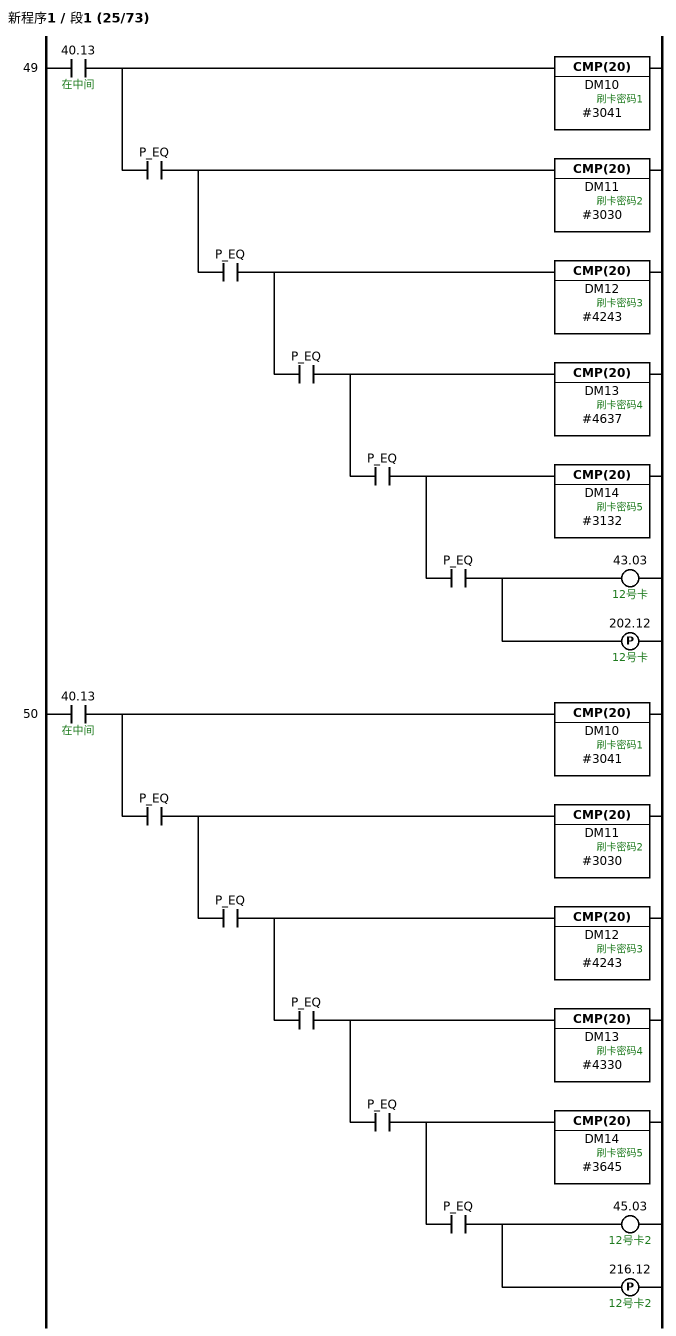
; [picture p24: 新程序1 / 段1, rungs 49-50]
; rung 49
LD 40.13  ; 在中间
CMP(20) DM10 #3041  ; 刷卡密码1
AND P_EQ
CMP(20) DM11 #3030  ; 刷卡密码2
AND P_EQ
CMP(20) DM12 #4243  ; 刷卡密码3
AND P_EQ
CMP(20) DM13 #4637  ; 刷卡密码4
AND P_EQ
CMP(20) DM14 #3132  ; 刷卡密码5
AND P_EQ
OUT 43.03  ; 12号卡
DIFU(13) 202.12  ; 12号卡
; rung 50
LD 40.13  ; 在中间
CMP(20) DM10 #3041  ; 刷卡密码1
AND P_EQ
CMP(20) DM11 #3030  ; 刷卡密码2
AND P_EQ
CMP(20) DM12 #4243  ; 刷卡密码3
AND P_EQ
CMP(20) DM13 #4330  ; 刷卡密码4
AND P_EQ
CMP(20) DM14 #3645  ; 刷卡密码5
AND P_EQ
OUT 45.03  ; 12号卡2
DIFU(13) 216.12  ; 12号卡2

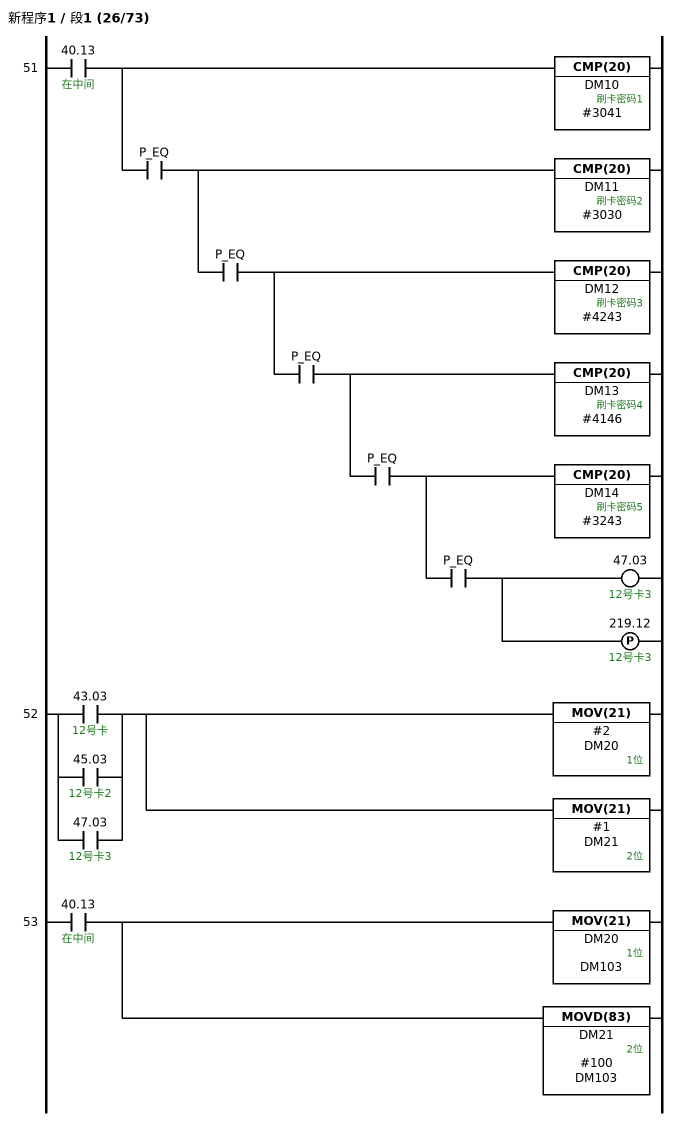
; rung 51
LD 40.13  ; 在中间
CMP(20) DM10 #3041  ; 刷卡密码1
AND P_EQ
CMP(20) DM11 #3030  ; 刷卡密码2
AND P_EQ
CMP(20) DM12 #4243  ; 刷卡密码3
AND P_EQ
CMP(20) DM13 #4146  ; 刷卡密码4
AND P_EQ
CMP(20) DM14 #3243  ; 刷卡密码5
AND P_EQ
OUT 47.03  ; 12号卡3
DIFU(13) 219.12  ; 12号卡3
; rung 52
LD 43.03  ; 12号卡
OR 45.03  ; 12号卡2
OR 47.03  ; 12号卡3
MOV(21) #2 DM20  ; 1位
MOV(21) #1 DM21  ; 2位
; rung 53
LD 40.13  ; 在中间
MOV(21) DM20 DM103  ; 1位
MOVD(83) DM21 #100 DM103  ; 2位

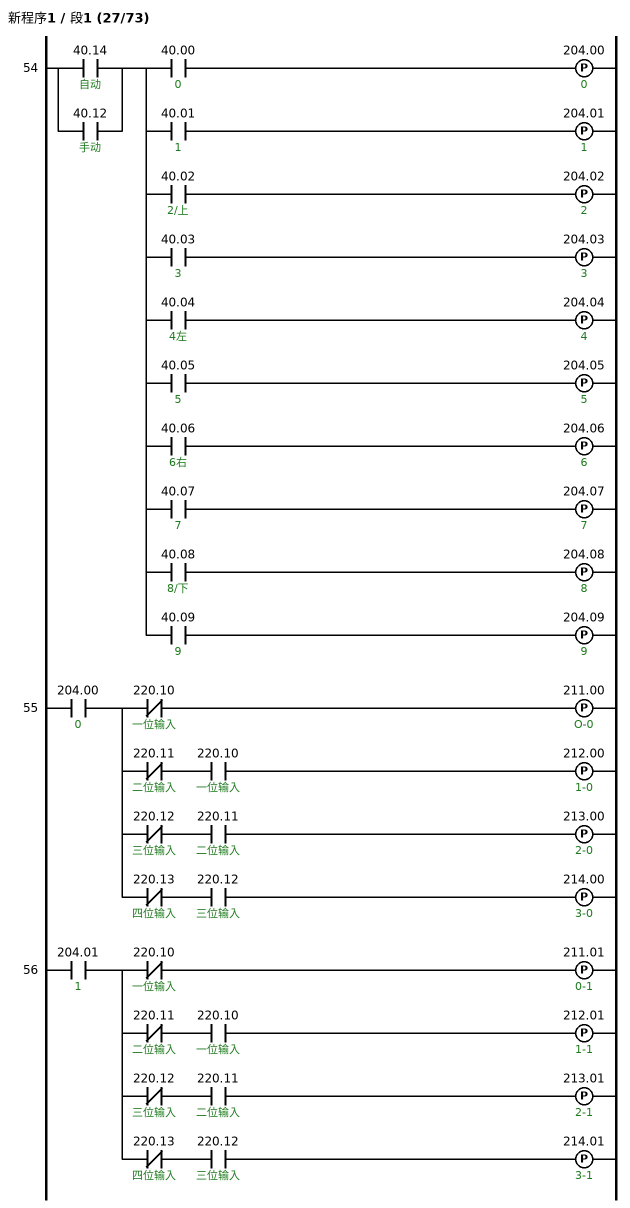
; rung 54
LD 40.14  ; 自动
OR 40.12  ; 手动
OUT TR0
AND 40.00  ; 0
DIFU(13) 204.00  ; 0
LD TR0
AND 40.01  ; 1
DIFU(13) 204.01  ; 1
LD TR0
AND 40.02  ; 2/上
DIFU(13) 204.02  ; 2
LD TR0
AND 40.03  ; 3
DIFU(13) 204.03  ; 3
LD TR0
AND 40.04  ; 4左
DIFU(13) 204.04  ; 4
LD TR0
AND 40.05  ; 5
DIFU(13) 204.05  ; 5
LD TR0
AND 40.06  ; 6右
DIFU(13) 204.06  ; 6
LD TR0
AND 40.07  ; 7
DIFU(13) 204.07  ; 7
LD TR0
AND 40.08  ; 8/下
DIFU(13) 204.08  ; 8
LD TR0
AND 40.09  ; 9
DIFU(13) 204.09  ; 9
; rung 55
LD 204.00  ; 0
OUT TR0
ANDNOT 220.10  ; 一位输入
DIFU(13) 211.00  ; O-0
LD TR0
ANDNOT 220.11  ; 二位输入
AND 220.10  ; 一位输入
DIFU(13) 212.00  ; 1-0
LD TR0
ANDNOT 220.12  ; 三位输入
AND 220.11  ; 二位输入
DIFU(13) 213.00  ; 2-0
LD TR0
ANDNOT 220.13  ; 四位输入
AND 220.12  ; 三位输入
DIFU(13) 214.00  ; 3-0
; rung 56
LD 204.01  ; 1
OUT TR0
ANDNOT 220.10  ; 一位输入
DIFU(13) 211.01  ; 0-1
LD TR0
ANDNOT 220.11  ; 二位输入
AND 220.10  ; 一位输入
DIFU(13) 212.01  ; 1-1
LD TR0
ANDNOT 220.12  ; 三位输入
AND 220.11  ; 二位输入
DIFU(13) 213.01  ; 2-1
LD TR0
ANDNOT 220.13  ; 四位输入
AND 220.12  ; 三位输入
DIFU(13) 214.01  ; 3-1

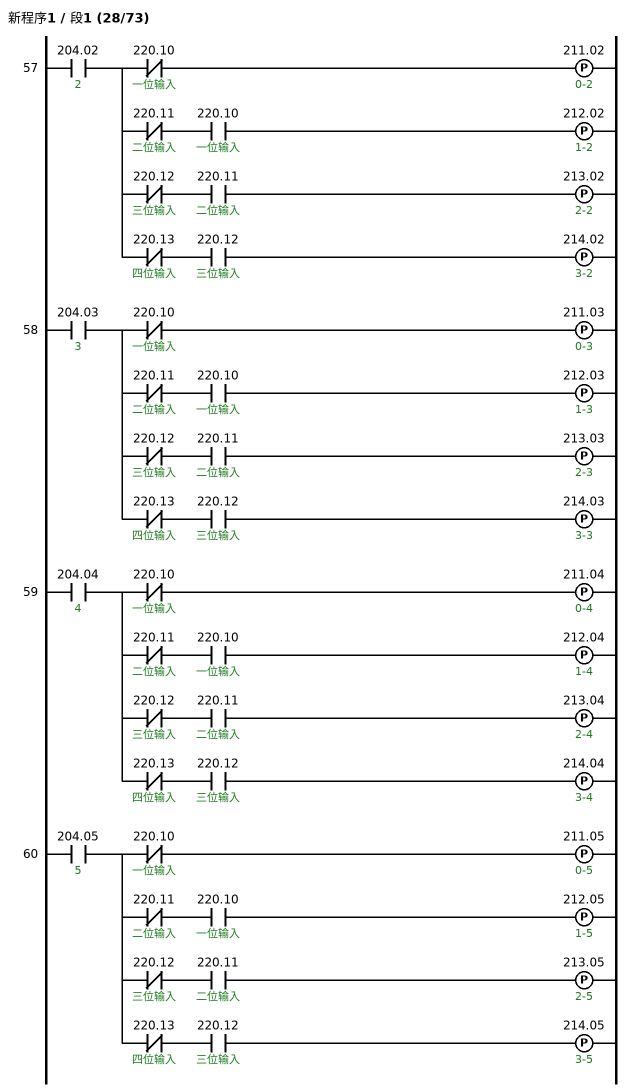
; rung 57
LD 204.02  ; 2
OUT TR0
ANDNOT 220.10  ; 一位输入
DIFU(13) 211.02  ; 0-2
LD TR0
ANDNOT 220.11  ; 二位输入
AND 220.10  ; 一位输入
DIFU(13) 212.02  ; 1-2
LD TR0
ANDNOT 220.12  ; 三位输入
AND 220.11  ; 二位输入
DIFU(13) 213.02  ; 2-2
LD TR0
ANDNOT 220.13  ; 四位输入
AND 220.12  ; 三位输入
DIFU(13) 214.02  ; 3-2
; rung 58
LD 204.03  ; 3
OUT TR0
ANDNOT 220.10  ; 一位输入
DIFU(13) 211.03  ; 0-3
LD TR0
ANDNOT 220.11  ; 二位输入
AND 220.10  ; 一位输入
DIFU(13) 212.03  ; 1-3
LD TR0
ANDNOT 220.12  ; 三位输入
AND 220.11  ; 二位输入
DIFU(13) 213.03  ; 2-3
LD TR0
ANDNOT 220.13  ; 四位输入
AND 220.12  ; 三位输入
DIFU(13) 214.03  ; 3-3
; rung 59
LD 204.04  ; 4
OUT TR0
ANDNOT 220.10  ; 一位输入
DIFU(13) 211.04  ; 0-4
LD TR0
ANDNOT 220.11  ; 二位输入
AND 220.10  ; 一位输入
DIFU(13) 212.04  ; 1-4
LD TR0
ANDNOT 220.12  ; 三位输入
AND 220.11  ; 二位输入
DIFU(13) 213.04  ; 2-4
LD TR0
ANDNOT 220.13  ; 四位输入
AND 220.12  ; 三位输入
DIFU(13) 214.04  ; 3-4
; rung 60
LD 204.05  ; 5
OUT TR0
ANDNOT 220.10  ; 一位输入
DIFU(13) 211.05  ; 0-5
LD TR0
ANDNOT 220.11  ; 二位输入
AND 220.10  ; 一位输入
DIFU(13) 212.05  ; 1-5
LD TR0
ANDNOT 220.12  ; 三位输入
AND 220.11  ; 二位输入
DIFU(13) 213.05  ; 2-5
LD TR0
ANDNOT 220.13  ; 四位输入
AND 220.12  ; 三位输入
DIFU(13) 214.05  ; 3-5

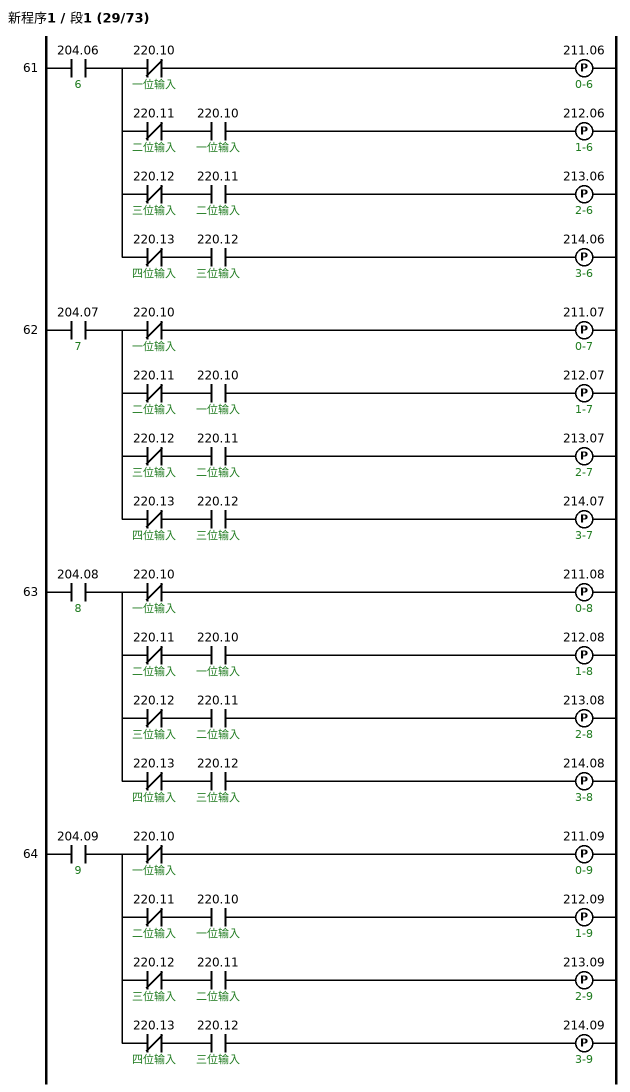
; rung 61
LD 204.06  ; 6
OUT TR0
ANDNOT 220.10  ; 一位输入
DIFU(13) 211.06  ; 0-6
LD TR0
ANDNOT 220.11  ; 二位输入
AND 220.10  ; 一位输入
DIFU(13) 212.06  ; 1-6
LD TR0
ANDNOT 220.12  ; 三位输入
AND 220.11  ; 二位输入
DIFU(13) 213.06  ; 2-6
LD TR0
ANDNOT 220.13  ; 四位输入
AND 220.12  ; 三位输入
DIFU(13) 214.06  ; 3-6
; rung 62
LD 204.07  ; 7
OUT TR0
ANDNOT 220.10  ; 一位输入
DIFU(13) 211.07  ; 0-7
LD TR0
ANDNOT 220.11  ; 二位输入
AND 220.10  ; 一位输入
DIFU(13) 212.07  ; 1-7
LD TR0
ANDNOT 220.12  ; 三位输入
AND 220.11  ; 二位输入
DIFU(13) 213.07  ; 2-7
LD TR0
ANDNOT 220.13  ; 四位输入
AND 220.12  ; 三位输入
DIFU(13) 214.07  ; 3-7
; rung 63
LD 204.08  ; 8
OUT TR0
ANDNOT 220.10  ; 一位输入
DIFU(13) 211.08  ; 0-8
LD TR0
ANDNOT 220.11  ; 二位输入
AND 220.10  ; 一位输入
DIFU(13) 212.08  ; 1-8
LD TR0
ANDNOT 220.12  ; 三位输入
AND 220.11  ; 二位输入
DIFU(13) 213.08  ; 2-8
LD TR0
ANDNOT 220.13  ; 四位输入
AND 220.12  ; 三位输入
DIFU(13) 214.08  ; 3-8
; rung 64
LD 204.09  ; 9
OUT TR0
ANDNOT 220.10  ; 一位输入
DIFU(13) 211.09  ; 0-9
LD TR0
ANDNOT 220.11  ; 二位输入
AND 220.10  ; 一位输入
DIFU(13) 212.09  ; 1-9
LD TR0
ANDNOT 220.12  ; 三位输入
AND 220.11  ; 二位输入
DIFU(13) 213.09  ; 2-9
LD TR0
ANDNOT 220.13  ; 四位输入
AND 220.12  ; 三位输入
DIFU(13) 214.09  ; 3-9

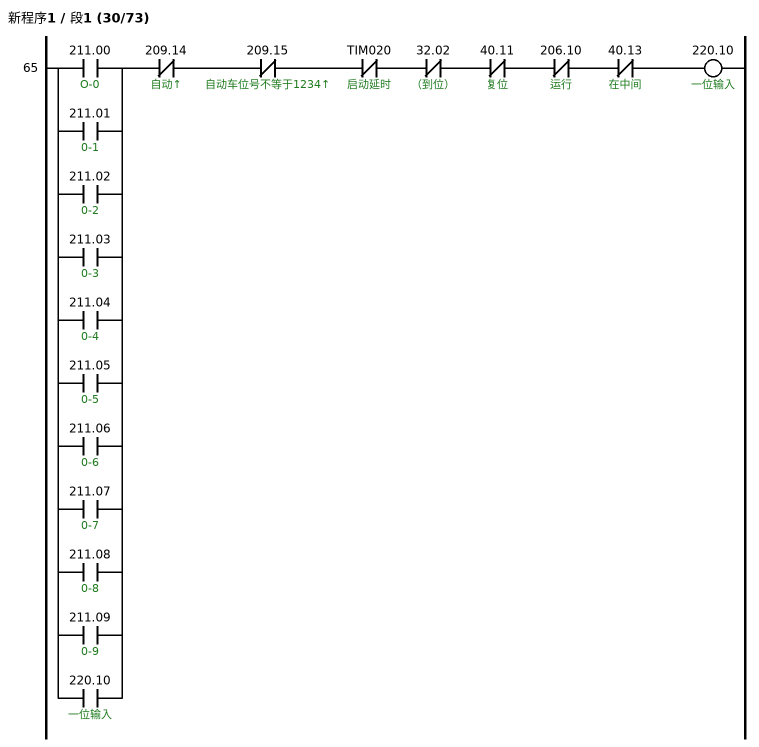
; rung 65
LD 211.00  ; O-0
OR 211.01  ; 0-1
OR 211.02  ; 0-2
OR 211.03  ; 0-3
OR 211.04  ; 0-4
OR 211.05  ; 0-5
OR 211.06  ; 0-6
OR 211.07  ; 0-7
OR 211.08  ; 0-8
OR 211.09  ; 0-9
OR 220.10  ; 一位输入
ANDNOT 209.14  ; 自动↑
ANDNOT 209.15  ; 自动车位号不等于1234↑
ANDNOT TIM020  ; 启动延时
ANDNOT 32.02  ; （到位）
ANDNOT 40.11  ; 复位
ANDNOT 206.10  ; 运行
ANDNOT 40.13  ; 在中间
OUT 220.10  ; 一位输入

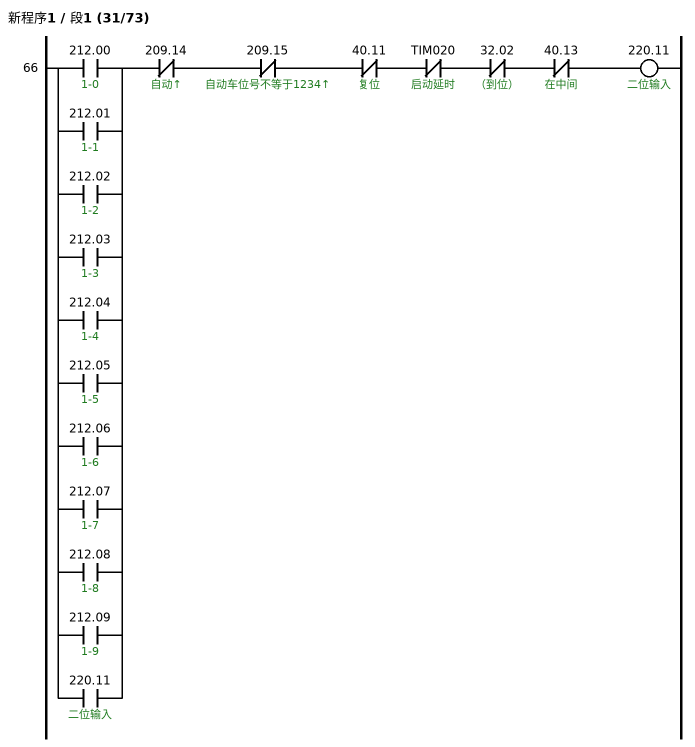
; rung 66
LD 212.00  ; 1-0
OR 212.01  ; 1-1
OR 212.02  ; 1-2
OR 212.03  ; 1-3
OR 212.04  ; 1-4
OR 212.05  ; 1-5
OR 212.06  ; 1-6
OR 212.07  ; 1-7
OR 212.08  ; 1-8
OR 212.09  ; 1-9
OR 220.11  ; 二位输入
ANDNOT 209.14  ; 自动↑
ANDNOT 209.15  ; 自动车位号不等于1234↑
ANDNOT 40.11  ; 复位
ANDNOT TIM020  ; 启动延时
ANDNOT 32.02  ; （到位）
ANDNOT 40.13  ; 在中间
OUT 220.11  ; 二位输入

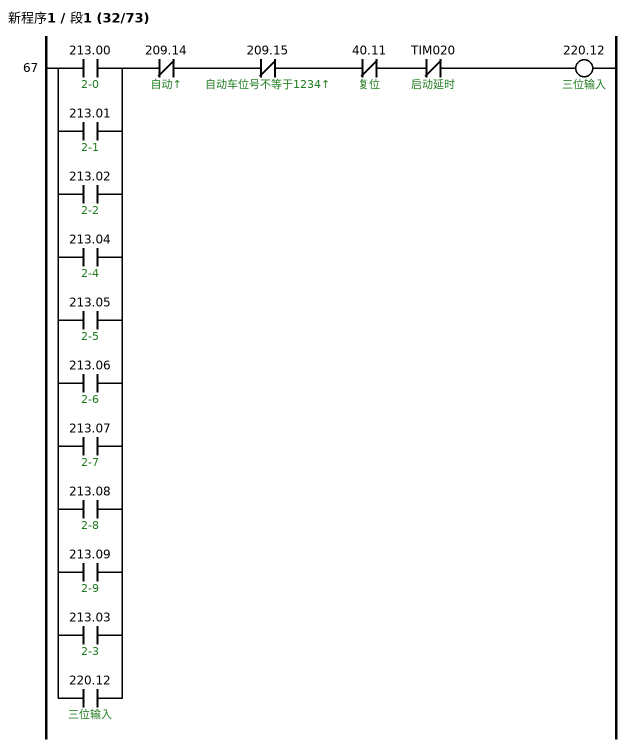
; rung 67
LD 213.00  ; 2-0
OR 213.01  ; 2-1
OR 213.02  ; 2-2
OR 213.04  ; 2-4
OR 213.05  ; 2-5
OR 213.06  ; 2-6
OR 213.07  ; 2-7
OR 213.08  ; 2-8
OR 213.09  ; 2-9
OR 213.03  ; 2-3
OR 220.12  ; 三位输入
ANDNOT 209.14  ; 自动↑
ANDNOT 209.15  ; 自动车位号不等于1234↑
ANDNOT 40.11  ; 复位
ANDNOT TIM020  ; 启动延时
OUT 220.12  ; 三位输入

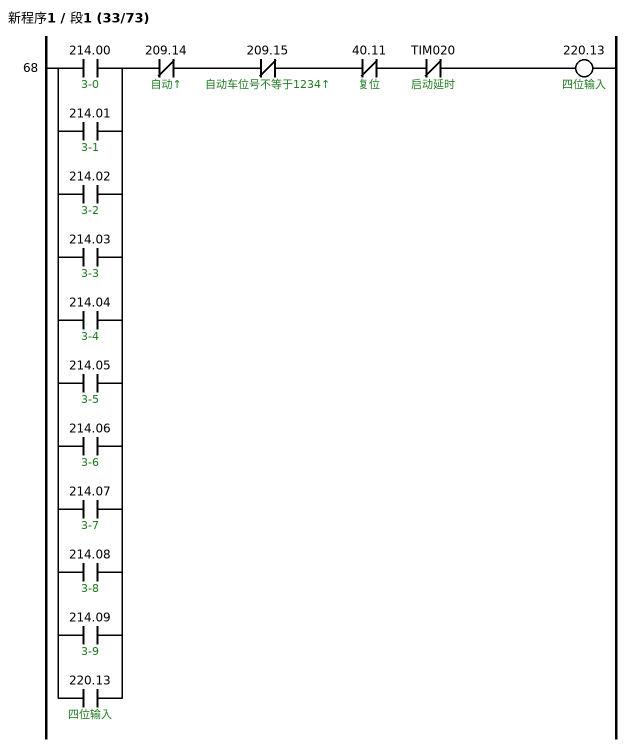
; rung 68
LD 214.00  ; 3-0
OR 214.01  ; 3-1
OR 214.02  ; 3-2
OR 214.03  ; 3-3
OR 214.04  ; 3-4
OR 214.05  ; 3-5
OR 214.06  ; 3-6
OR 214.07  ; 3-7
OR 214.08  ; 3-8
OR 214.09  ; 3-9
OR 220.13  ; 四位输入
ANDNOT 209.14  ; 自动↑
ANDNOT 209.15  ; 自动车位号不等于1234↑
ANDNOT 40.11  ; 复位
ANDNOT TIM020  ; 启动延时
OUT 220.13  ; 四位输入

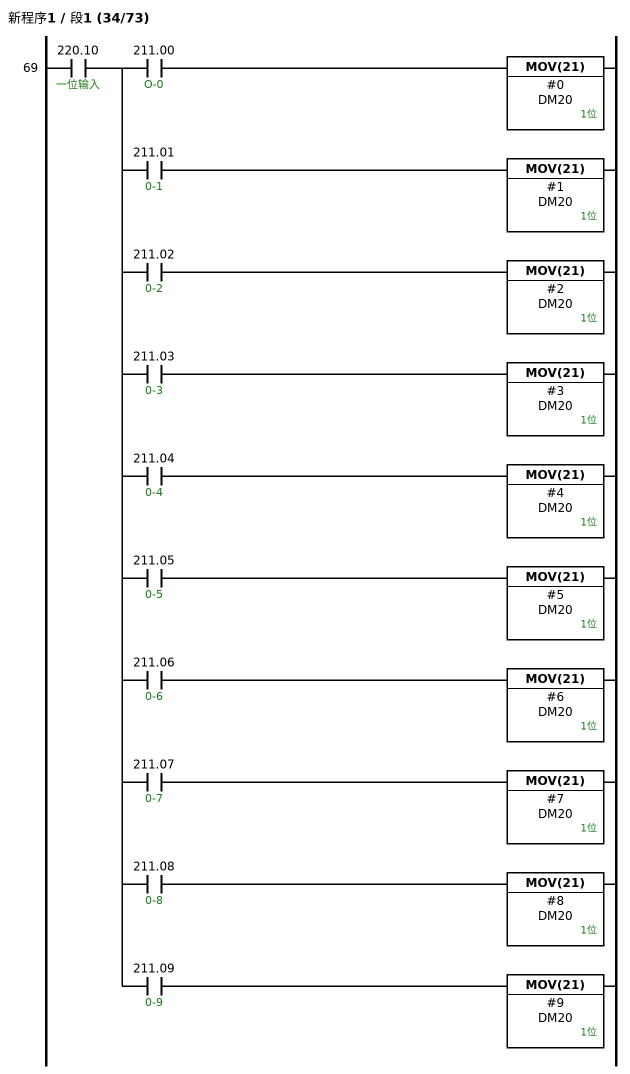
; rung 69
LD 220.10  ; 一位输入
OUT TR0
AND 211.00  ; O-0
MOV(21) #0 DM20  ; 1位
LD TR0
AND 211.01  ; 0-1
MOV(21) #1 DM20  ; 1位
LD TR0
AND 211.02  ; 0-2
MOV(21) #2 DM20  ; 1位
LD TR0
AND 211.03  ; 0-3
MOV(21) #3 DM20  ; 1位
LD TR0
AND 211.04  ; 0-4
MOV(21) #4 DM20  ; 1位
LD TR0
AND 211.05  ; 0-5
MOV(21) #5 DM20  ; 1位
LD TR0
AND 211.06  ; 0-6
MOV(21) #6 DM20  ; 1位
LD TR0
AND 211.07  ; 0-7
MOV(21) #7 DM20  ; 1位
LD TR0
AND 211.08  ; 0-8
MOV(21) #8 DM20  ; 1位
LD TR0
AND 211.09  ; 0-9
MOV(21) #9 DM20  ; 1位

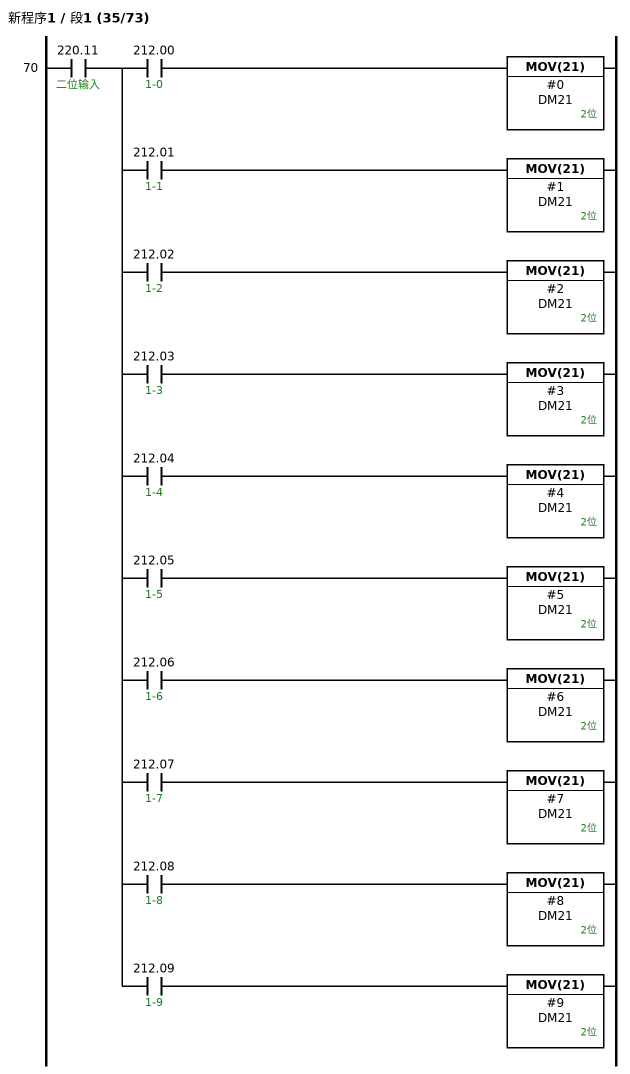
; rung 70
LD 220.11  ; 二位输入
OUT TR0
AND 212.00  ; 1-0
MOV(21) #0 DM21  ; 2位
LD TR0
AND 212.01  ; 1-1
MOV(21) #1 DM21  ; 2位
LD TR0
AND 212.02  ; 1-2
MOV(21) #2 DM21  ; 2位
LD TR0
AND 212.03  ; 1-3
MOV(21) #3 DM21  ; 2位
LD TR0
AND 212.04  ; 1-4
MOV(21) #4 DM21  ; 2位
LD TR0
AND 212.05  ; 1-5
MOV(21) #5 DM21  ; 2位
LD TR0
AND 212.06  ; 1-6
MOV(21) #6 DM21  ; 2位
LD TR0
AND 212.07  ; 1-7
MOV(21) #7 DM21  ; 2位
LD TR0
AND 212.08  ; 1-8
MOV(21) #8 DM21  ; 2位
LD TR0
AND 212.09  ; 1-9
MOV(21) #9 DM21  ; 2位

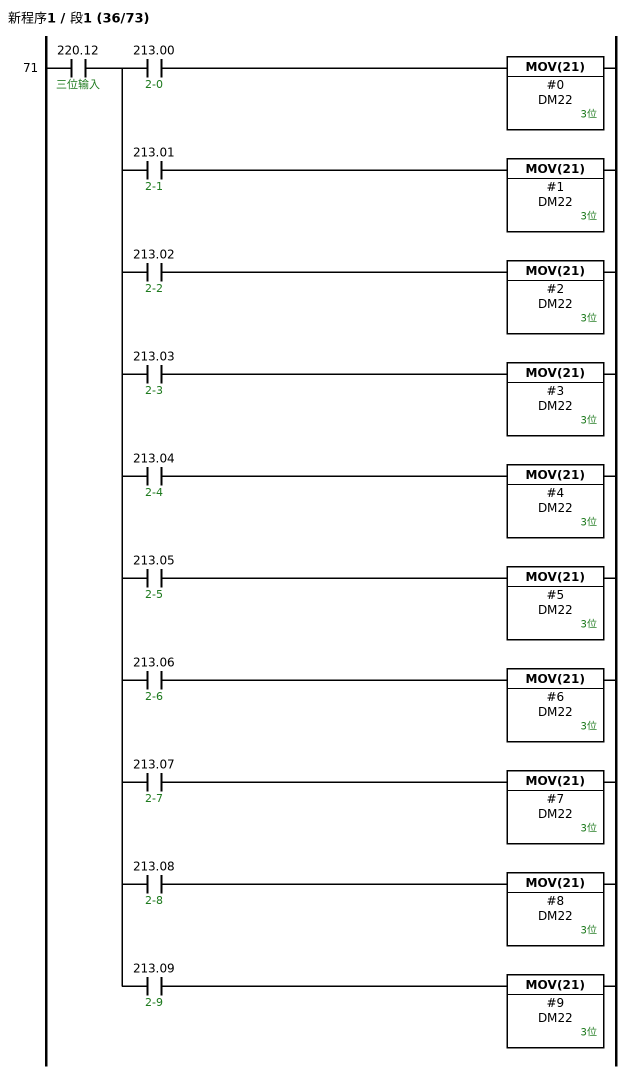
; rung 71
LD 220.12  ; 三位输入
OUT TR0
AND 213.00  ; 2-0
MOV(21) #0 DM22  ; 3位
LD TR0
AND 213.01  ; 2-1
MOV(21) #1 DM22  ; 3位
LD TR0
AND 213.02  ; 2-2
MOV(21) #2 DM22  ; 3位
LD TR0
AND 213.03  ; 2-3
MOV(21) #3 DM22  ; 3位
LD TR0
AND 213.04  ; 2-4
MOV(21) #4 DM22  ; 3位
LD TR0
AND 213.05  ; 2-5
MOV(21) #5 DM22  ; 3位
LD TR0
AND 213.06  ; 2-6
MOV(21) #6 DM22  ; 3位
LD TR0
AND 213.07  ; 2-7
MOV(21) #7 DM22  ; 3位
LD TR0
AND 213.08  ; 2-8
MOV(21) #8 DM22  ; 3位
LD TR0
AND 213.09  ; 2-9
MOV(21) #9 DM22  ; 3位

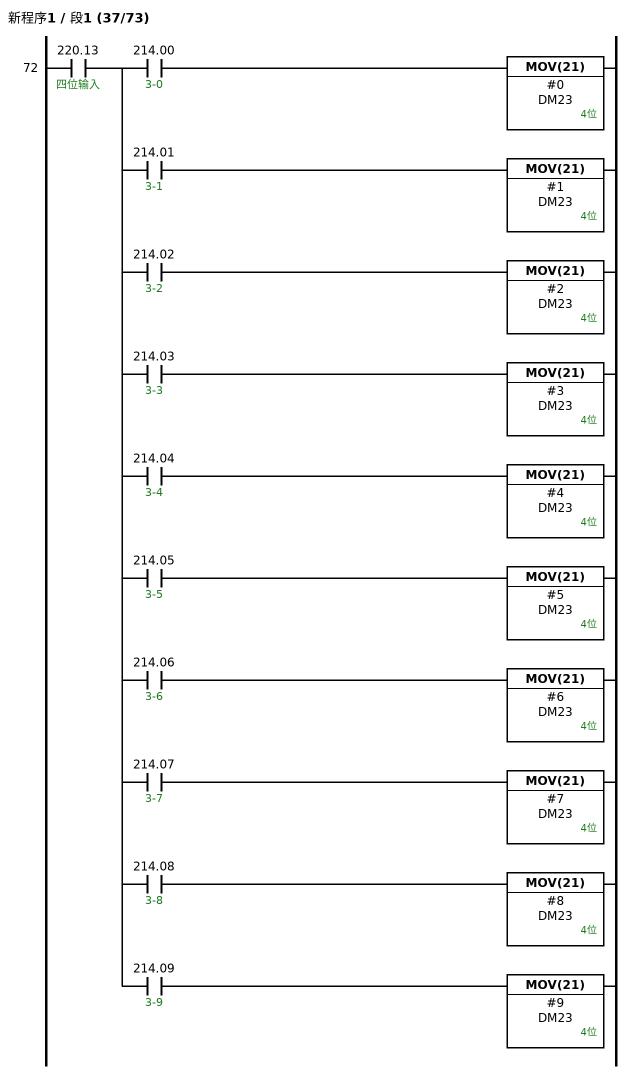
; rung 72
LD 220.13  ; 四位输入
OUT TR0
AND 214.00  ; 3-0
MOV(21) #0 DM23  ; 4位
LD TR0
AND 214.01  ; 3-1
MOV(21) #1 DM23  ; 4位
LD TR0
AND 214.02  ; 3-2
MOV(21) #2 DM23  ; 4位
LD TR0
AND 214.03  ; 3-3
MOV(21) #3 DM23  ; 4位
LD TR0
AND 214.04  ; 3-4
MOV(21) #4 DM23  ; 4位
LD TR0
AND 214.05  ; 3-5
MOV(21) #5 DM23  ; 4位
LD TR0
AND 214.06  ; 3-6
MOV(21) #6 DM23  ; 4位
LD TR0
AND 214.07  ; 3-7
MOV(21) #7 DM23  ; 4位
LD TR0
AND 214.08  ; 3-8
MOV(21) #8 DM23  ; 4位
LD TR0
AND 214.09  ; 3-9
MOV(21) #9 DM23  ; 4位

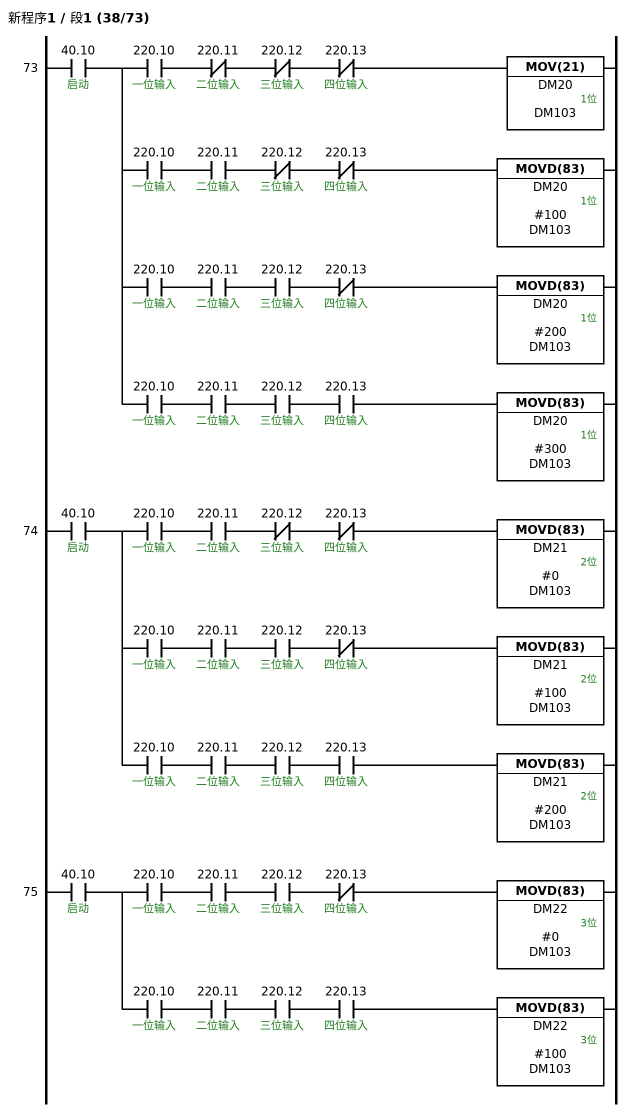
; rung 73
LD 40.10  ; 启动
OUT TR0
AND 220.10  ; 一位输入
ANDNOT 220.11  ; 二位输入
ANDNOT 220.12  ; 三位输入
ANDNOT 220.13  ; 四位输入
MOV(21) DM20 DM103  ; 1位
LD TR0
AND 220.10  ; 一位输入
AND 220.11  ; 二位输入
ANDNOT 220.12  ; 三位输入
ANDNOT 220.13  ; 四位输入
MOVD(83) DM20 #100 DM103  ; 1位
LD TR0
AND 220.10  ; 一位输入
AND 220.11  ; 二位输入
AND 220.12  ; 三位输入
ANDNOT 220.13  ; 四位输入
MOVD(83) DM20 #200 DM103  ; 1位
LD TR0
AND 220.10  ; 一位输入
AND 220.11  ; 二位输入
AND 220.12  ; 三位输入
AND 220.13  ; 四位输入
MOVD(83) DM20 #300 DM103  ; 1位
; rung 74
LD 40.10  ; 启动
OUT TR0
AND 220.10  ; 一位输入
AND 220.11  ; 二位输入
ANDNOT 220.12  ; 三位输入
ANDNOT 220.13  ; 四位输入
MOVD(83) DM21 #0 DM103  ; 2位
LD TR0
AND 220.10  ; 一位输入
AND 220.11  ; 二位输入
AND 220.12  ; 三位输入
ANDNOT 220.13  ; 四位输入
MOVD(83) DM21 #100 DM103  ; 2位
LD TR0
AND 220.10  ; 一位输入
AND 220.11  ; 二位输入
AND 220.12  ; 三位输入
AND 220.13  ; 四位输入
MOVD(83) DM21 #200 DM103  ; 2位
; rung 75
LD 40.10  ; 启动
OUT TR0
AND 220.10  ; 一位输入
AND 220.11  ; 二位输入
AND 220.12  ; 三位输入
ANDNOT 220.13  ; 四位输入
MOVD(83) DM22 #0 DM103  ; 3位
LD TR0
AND 220.10  ; 一位输入
AND 220.11  ; 二位输入
AND 220.12  ; 三位输入
AND 220.13  ; 四位输入
MOVD(83) DM22 #100 DM103  ; 3位

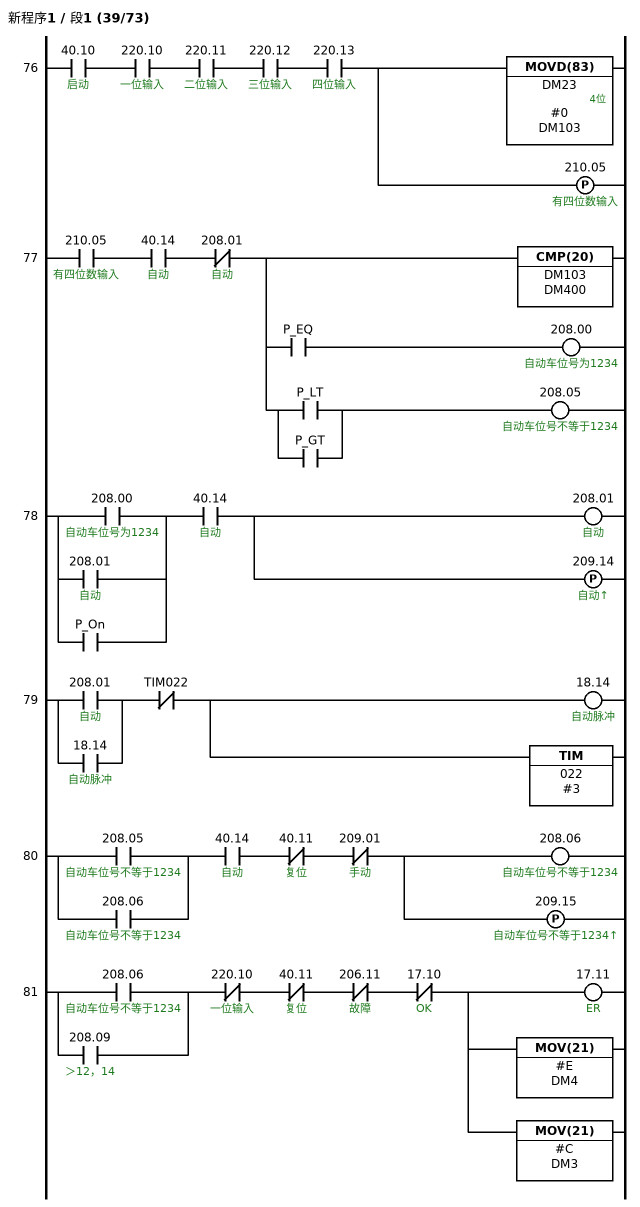
; rung 76
LD 40.10  ; 启动
AND 220.10  ; 一位输入
AND 220.11  ; 二位输入
AND 220.12  ; 三位输入
AND 220.13  ; 四位输入
MOVD(83) DM23 #0 DM103  ; 4位
DIFU(13) 210.05  ; 有四位数输入
; rung 77
LD 210.05  ; 有四位数输入
AND 40.14  ; 自动
ANDNOT 208.01  ; 自动
OUT TR0
CMP(20) DM103 DM400
AND P_EQ
OUT 208.00  ; 自动车位号为1234
LD TR0
LD P_LT
OR P_GT
ANDLD
OUT 208.05  ; 自动车位号不等于1234
; rung 78
LD 208.00  ; 自动车位号为1234
OR 208.01  ; 自动
OR P_On
AND 40.14  ; 自动
OUT 208.01  ; 自动
DIFU(13) 209.14  ; 自动↑
; rung 79
LD 208.01  ; 自动
OR 18.14  ; 自动脉冲
ANDNOT TIM022
OUT 18.14  ; 自动脉冲
TIM 022 #3
; rung 80
LD 208.05  ; 自动车位号不等于1234
OR 208.06  ; 自动车位号不等于1234
AND 40.14  ; 自动
ANDNOT 40.11  ; 复位
ANDNOT 209.01  ; 手动
OUT 208.06  ; 自动车位号不等于1234
DIFU(13) 209.15  ; 自动车位号不等于1234↑
; rung 81
LD 208.06  ; 自动车位号不等于1234
OR 208.09  ; ＞12，14
ANDNOT 220.10  ; 一位输入
ANDNOT 40.11  ; 复位
ANDNOT 206.11  ; 故障
ANDNOT 17.10  ; OK
OUT 17.11  ; ER
MOV(21) #E DM4
MOV(21) #C DM3

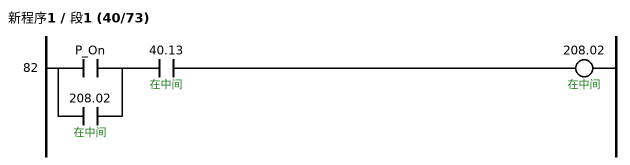
; rung 82
LD P_On
OR 208.02  ; 在中间
AND 40.13  ; 在中间
OUT 208.02  ; 在中间

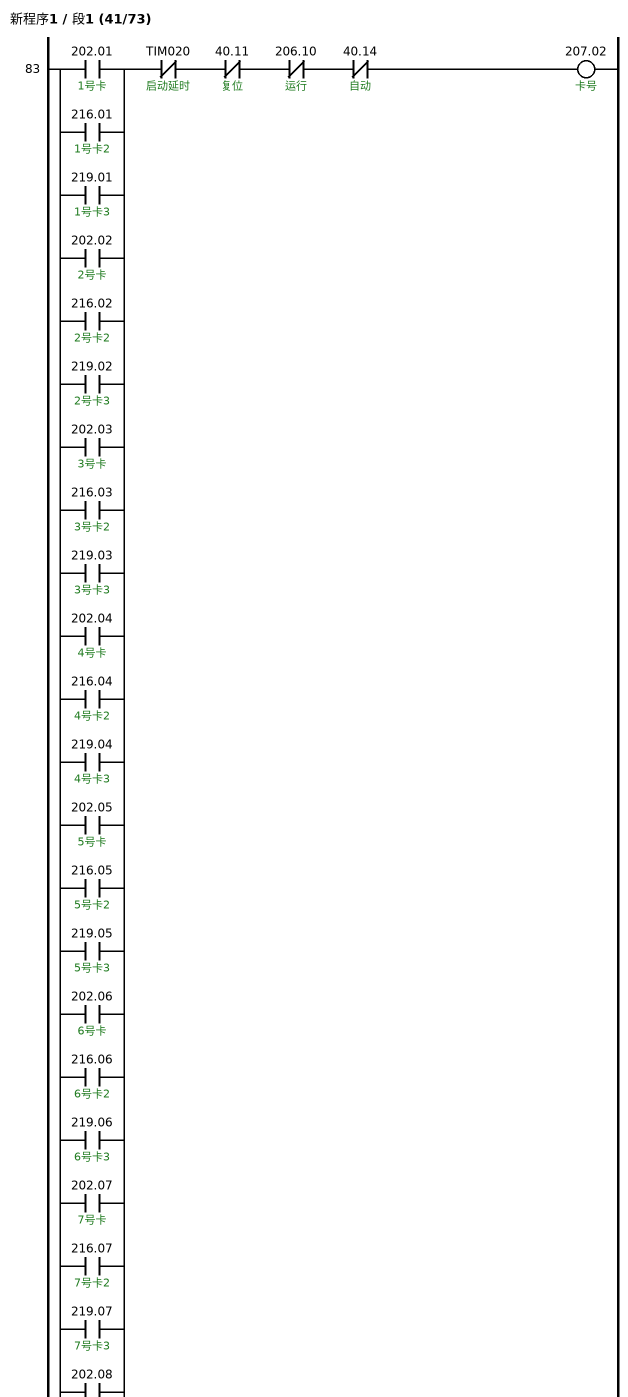

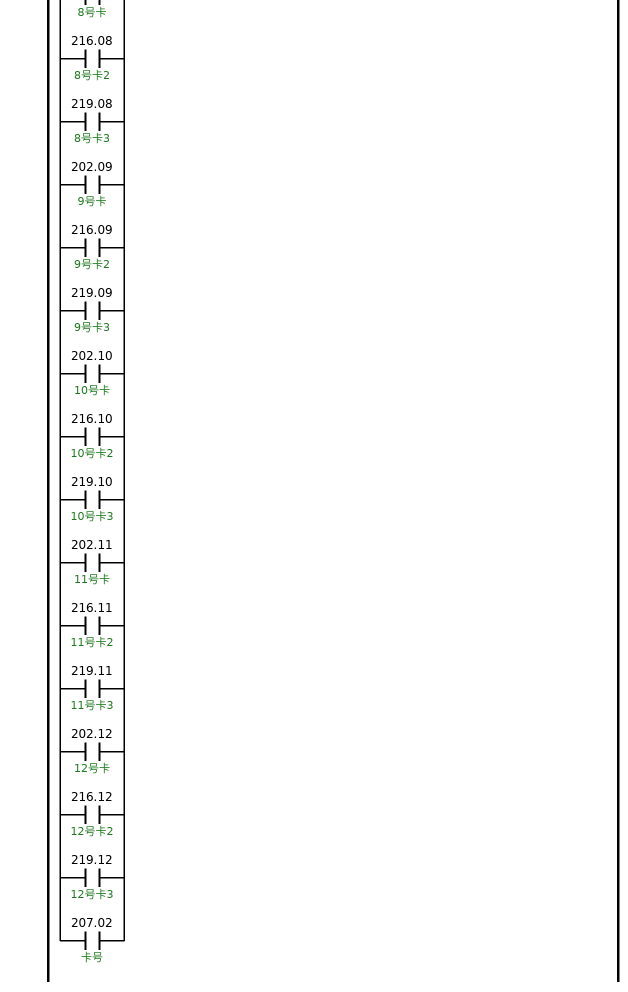
; rung 83
LD 202.01  ; 1号卡
OR 216.01  ; 1号卡2
OR 219.01  ; 1号卡3
OR 202.02  ; 2号卡
OR 216.02  ; 2号卡2
OR 219.02  ; 2号卡3
OR 202.03  ; 3号卡
OR 216.03  ; 3号卡2
OR 219.03  ; 3号卡3
OR 202.04  ; 4号卡
OR 216.04  ; 4号卡2
OR 219.04  ; 4号卡3
OR 202.05  ; 5号卡
OR 216.05  ; 5号卡2
OR 219.05  ; 5号卡3
OR 202.06  ; 6号卡
OR 216.06  ; 6号卡2
OR 219.06  ; 6号卡3
OR 202.07  ; 7号卡
OR 216.07  ; 7号卡2
OR 219.07  ; 7号卡3
OR 202.08  ; 8号卡
OR 216.08  ; 8号卡2
OR 219.08  ; 8号卡3
OR 202.09  ; 9号卡
OR 216.09  ; 9号卡2
OR 219.09  ; 9号卡3
OR 202.10  ; 10号卡
OR 216.10  ; 10号卡2
OR 219.10  ; 10号卡3
OR 202.11  ; 11号卡
OR 216.11  ; 11号卡2
OR 219.11  ; 11号卡3
OR 202.12  ; 12号卡
OR 216.12  ; 12号卡2
OR 219.12  ; 12号卡3
OR 207.02  ; 卡号
ANDNOT TIM020  ; 启动延时
ANDNOT 40.11  ; 复位
ANDNOT 206.10  ; 运行
ANDNOT 40.14  ; 自动
OUT 207.02  ; 卡号

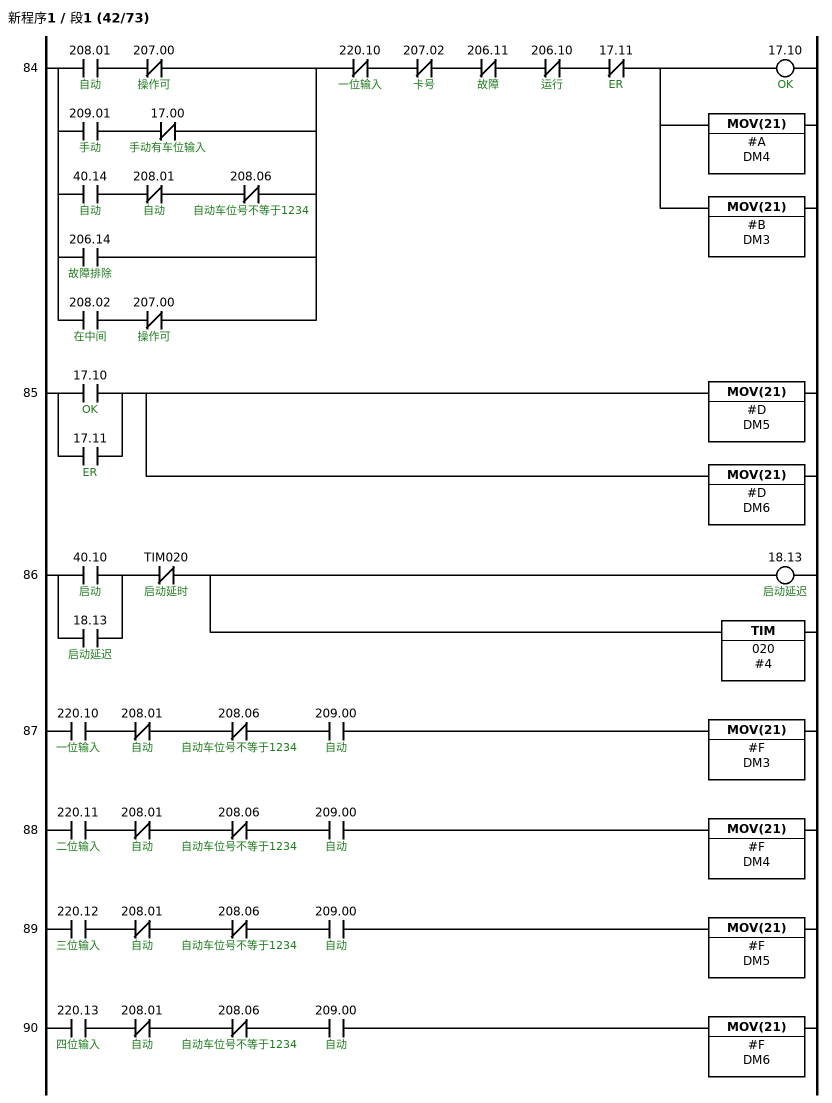
; rung 84
LD 208.01  ; 自动
ANDNOT 207.00  ; 操作可
LD 209.01  ; 手动
ANDNOT 17.00  ; 手动有车位输入
ORLD
LD 40.14  ; 自动
ANDNOT 208.01  ; 自动
ANDNOT 208.06  ; 自动车位号不等于1234
ORLD
OR 206.14  ; 故障排除
LD 208.02  ; 在中间
ANDNOT 207.00  ; 操作可
ORLD
ANDNOT 220.10  ; 一位输入
ANDNOT 207.02  ; 卡号
ANDNOT 206.11  ; 故障
ANDNOT 206.10  ; 运行
ANDNOT 17.11  ; ER
OUT 17.10  ; OK
MOV(21) #A DM4
MOV(21) #B DM3
; rung 85
LD 17.10  ; OK
OR 17.11  ; ER
MOV(21) #D DM5
MOV(21) #D DM6
; rung 86
LD 40.10  ; 启动
OR 18.13  ; 启动延迟
ANDNOT TIM020  ; 启动延时
OUT 18.13  ; 启动延迟
TIM 020 #4
; rung 87
LD 220.10  ; 一位输入
ANDNOT 208.01  ; 自动
ANDNOT 208.06  ; 自动车位号不等于1234
AND 209.00  ; 自动
MOV(21) #F DM3
; rung 88
LD 220.11  ; 二位输入
ANDNOT 208.01  ; 自动
ANDNOT 208.06  ; 自动车位号不等于1234
AND 209.00  ; 自动
MOV(21) #F DM4
; rung 89
LD 220.12  ; 三位输入
ANDNOT 208.01  ; 自动
ANDNOT 208.06  ; 自动车位号不等于1234
AND 209.00  ; 自动
MOV(21) #F DM5
; rung 90
LD 220.13  ; 四位输入
ANDNOT 208.01  ; 自动
ANDNOT 208.06  ; 自动车位号不等于1234
AND 209.00  ; 自动
MOV(21) #F DM6

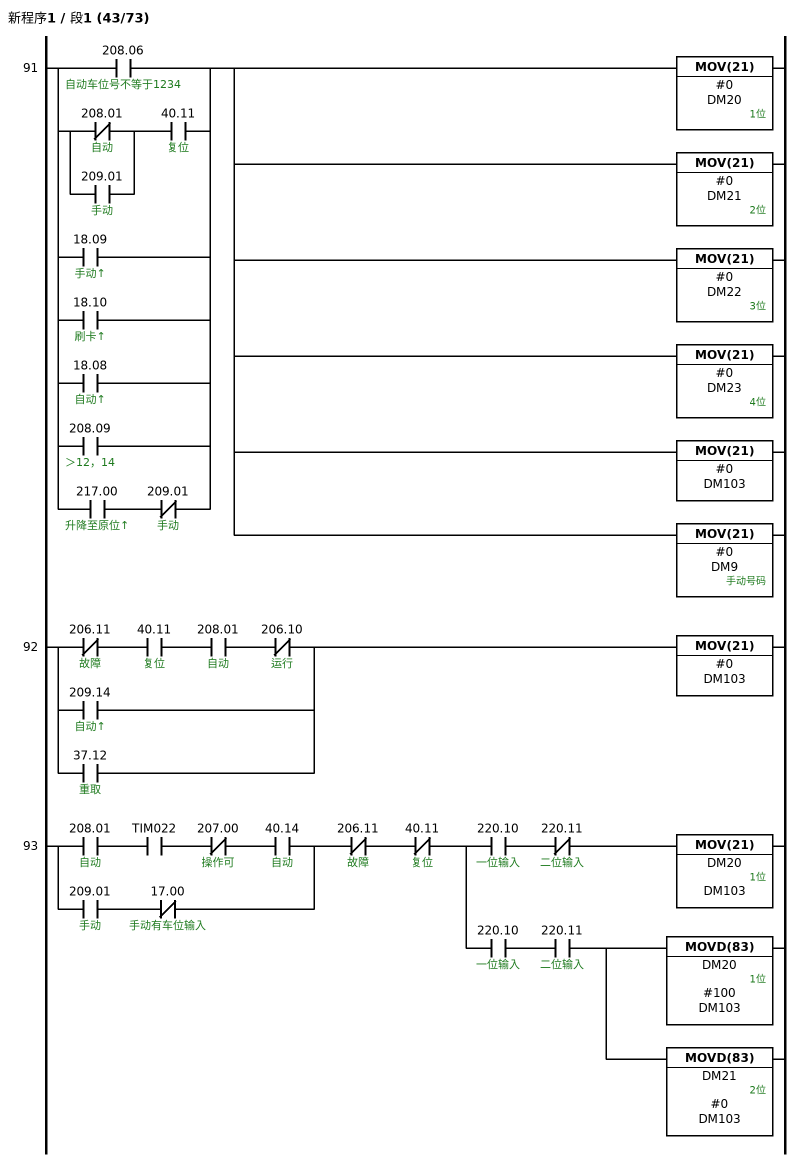
; rung 91
LD 208.06  ; 自动车位号不等于1234
LDNOT 208.01  ; 自动
OR 209.01  ; 手动
AND 40.11  ; 复位
ORLD
OR 18.09  ; 手动↑
OR 18.10  ; 刷卡↑
OR 18.08  ; 自动↑
OR 208.09  ; ＞12，14
LD 217.00  ; 升降至原位↑
ANDNOT 209.01  ; 手动
ORLD
MOV(21) #0 DM20  ; 1位
MOV(21) #0 DM21  ; 2位
MOV(21) #0 DM22  ; 3位
MOV(21) #0 DM23  ; 4位
MOV(21) #0 DM103
MOV(21) #0 DM9  ; 手动号码
; rung 92
LDNOT 206.11  ; 故障
AND 40.11  ; 复位
AND 208.01  ; 自动
ANDNOT 206.10  ; 运行
OR 209.14  ; 自动↑
OR 37.12  ; 重取
MOV(21) #0 DM103
; rung 93
LD 208.01  ; 自动
AND TIM022
ANDNOT 207.00  ; 操作可
AND 40.14  ; 自动
LD 209.01  ; 手动
ANDNOT 17.00  ; 手动有车位输入
ORLD
ANDNOT 206.11  ; 故障
ANDNOT 40.11  ; 复位
OUT TR0
AND 220.10  ; 一位输入
ANDNOT 220.11  ; 二位输入
MOV(21) DM20 DM103  ; 1位
LD TR0
AND 220.10  ; 一位输入
AND 220.11  ; 二位输入
MOVD(83) DM20 #100 DM103  ; 1位
MOVD(83) DM21 #0 DM103  ; 2位

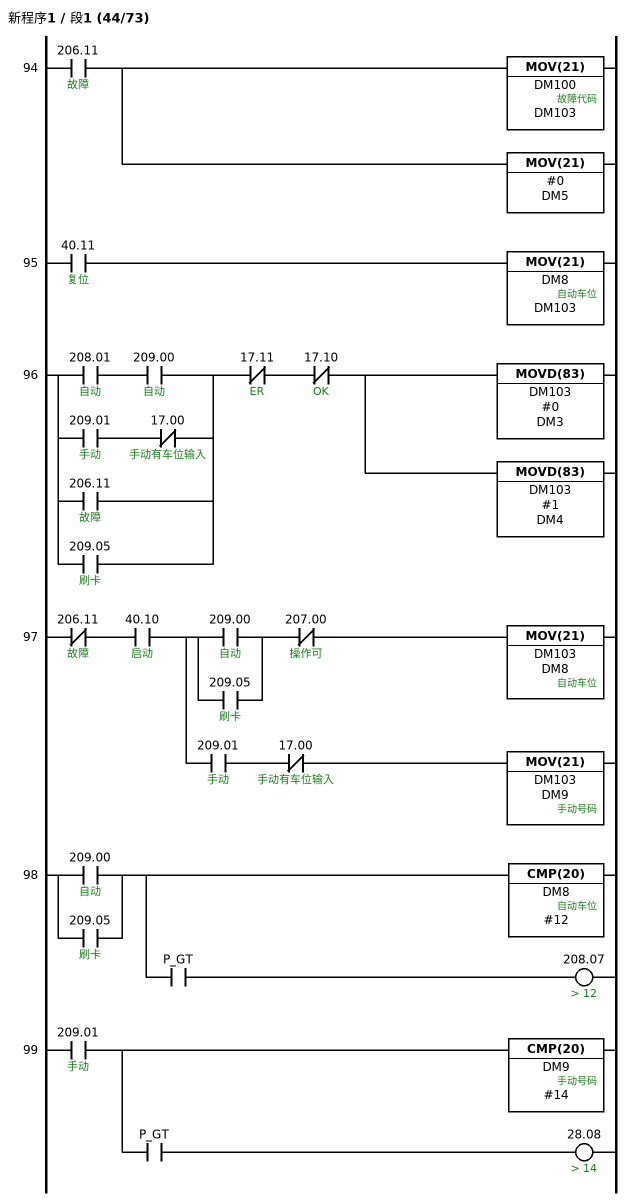
; rung 94
LD 206.11  ; 故障
MOV(21) DM100 DM103  ; 故障代码
MOV(21) #0 DM5
; rung 95
LD 40.11  ; 复位
MOV(21) DM8 DM103  ; 自动车位
; rung 96
LD 208.01  ; 自动
AND 209.00  ; 自动
LD 209.01  ; 手动
ANDNOT 17.00  ; 手动有车位输入
ORLD
OR 206.11  ; 故障
OR 209.05  ; 刷卡
ANDNOT 17.11  ; ER
ANDNOT 17.10  ; OK
MOVD(83) DM103 #0 DM3
MOVD(83) DM103 #1 DM4
; rung 97
LDNOT 206.11  ; 故障
AND 40.10  ; 启动
OUT TR0
LD 209.00  ; 自动
OR 209.05  ; 刷卡
ANDLD
ANDNOT 207.00  ; 操作可
MOV(21) DM103 DM8  ; 自动车位
LD TR0
AND 209.01  ; 手动
ANDNOT 17.00  ; 手动有车位输入
MOV(21) DM103 DM9  ; 手动号码
; rung 98
LD 209.00  ; 自动
OR 209.05  ; 刷卡
CMP(20) DM8 #12  ; 自动车位
AND P_GT
OUT 208.07  ; > 12
; rung 99
LD 209.01  ; 手动
CMP(20) DM9 #14  ; 手动号码
AND P_GT
OUT 28.08  ; > 14

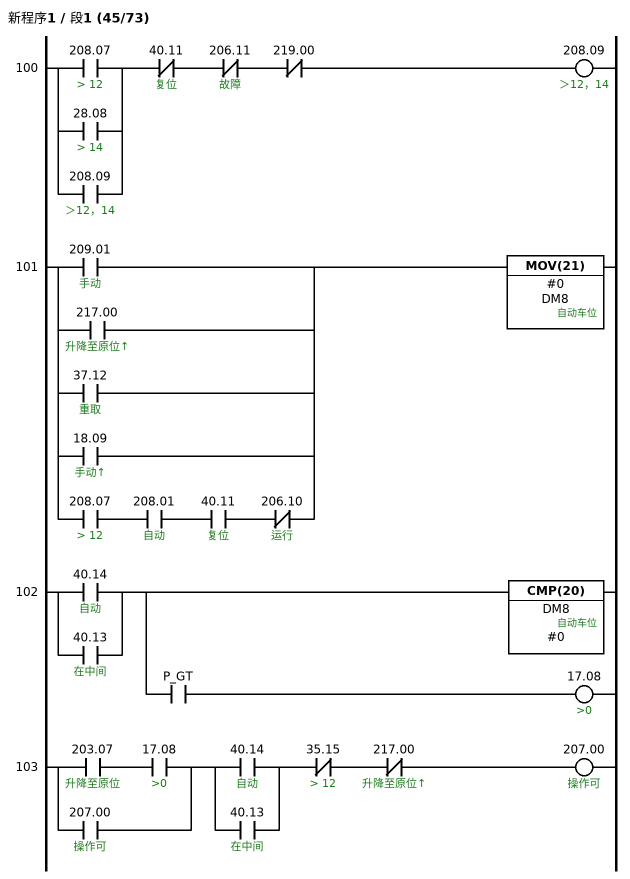
; rung 100
LD 208.07  ; > 12
OR 28.08  ; > 14
OR 208.09  ; ＞12，14
ANDNOT 40.11  ; 复位
ANDNOT 206.11  ; 故障
ANDNOT 219.00
OUT 208.09  ; ＞12，14
; rung 101
LD 209.01  ; 手动
OR 217.00  ; 升降至原位↑
OR 37.12  ; 重取
OR 18.09  ; 手动↑
LD 208.07  ; > 12
AND 208.01  ; 自动
AND 40.11  ; 复位
ANDNOT 206.10  ; 运行
ORLD
MOV(21) #0 DM8  ; 自动车位
; rung 102
LD 40.14  ; 自动
OR 40.13  ; 在中间
CMP(20) DM8 #0  ; 自动车位
AND P_GT
OUT 17.08  ; >0
; rung 103
LD 203.07  ; 升降至原位
AND 17.08  ; >0
OR 207.00  ; 操作可
LD 40.14  ; 自动
OR 40.13  ; 在中间
ANDLD
ANDNOT 35.15  ; > 12
ANDNOT 217.00  ; 升降至原位↑
OUT 207.00  ; 操作可

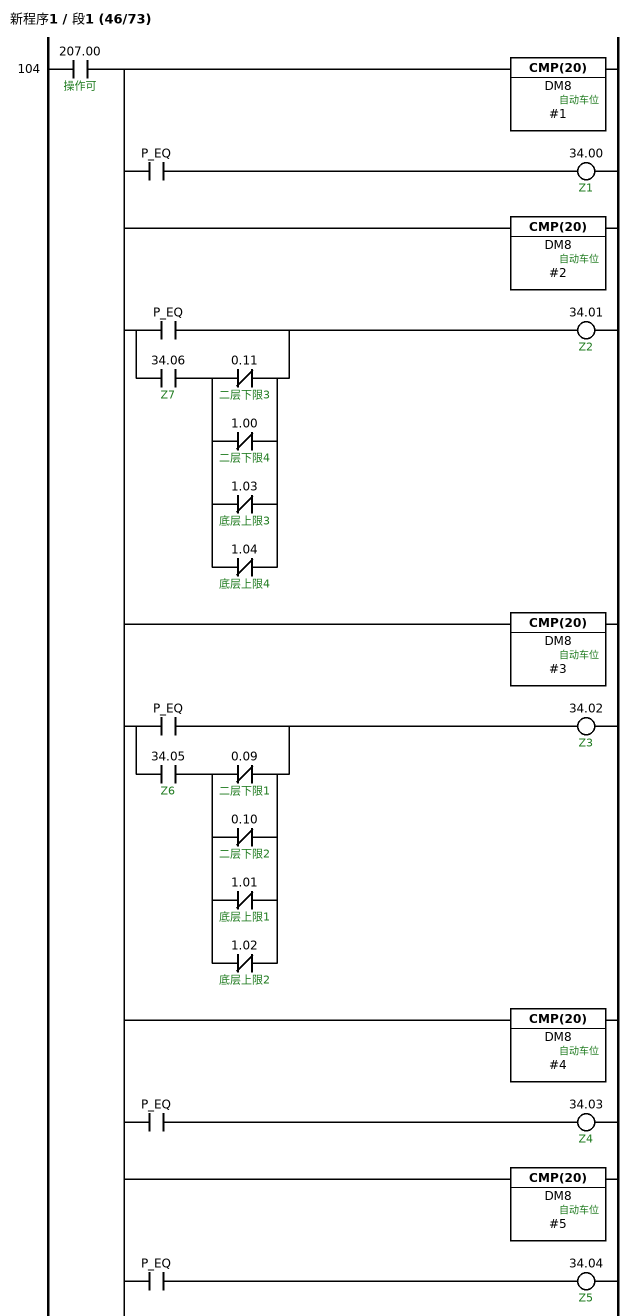

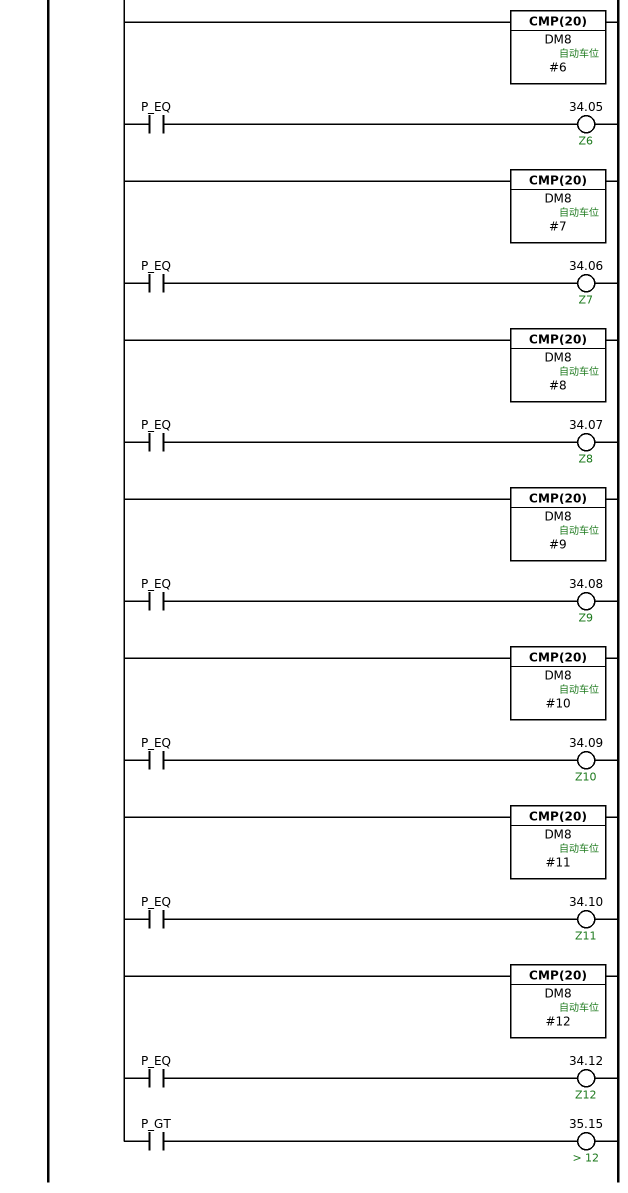
; rung 104
LD 207.00  ; 操作可
OUT TR0
CMP(20) DM8 #1  ; 自动车位
AND P_EQ
OUT 34.00  ; Z1
LD TR0
CMP(20) DM8 #2  ; 自动车位
LD P_EQ
LD 34.06  ; Z7
LDNOT 0.11  ; 二层下限3
ORNOT 1.00  ; 二层下限4
ORNOT 1.03  ; 底层上限3
ORNOT 1.04  ; 底层上限4
ANDLD
ORLD
ANDLD
OUT 34.01  ; Z2
LD TR0
CMP(20) DM8 #3  ; 自动车位
LD P_EQ
LD 34.05  ; Z6
LDNOT 0.09  ; 二层下限1
ORNOT 0.10  ; 二层下限2
ORNOT 1.01  ; 底层上限1
ORNOT 1.02  ; 底层上限2
ANDLD
ORLD
ANDLD
OUT 34.02  ; Z3
LD TR0
CMP(20) DM8 #4  ; 自动车位
AND P_EQ
OUT 34.03  ; Z4
LD TR0
CMP(20) DM8 #5  ; 自动车位
AND P_EQ
OUT 34.04  ; Z5
LD TR0
CMP(20) DM8 #6  ; 自动车位
AND P_EQ
OUT 34.05  ; Z6
LD TR0
CMP(20) DM8 #7  ; 自动车位
AND P_EQ
OUT 34.06  ; Z7
LD TR0
CMP(20) DM8 #8  ; 自动车位
AND P_EQ
OUT 34.07  ; Z8
LD TR0
CMP(20) DM8 #9  ; 自动车位
AND P_EQ
OUT 34.08  ; Z9
LD TR0
CMP(20) DM8 #10  ; 自动车位
AND P_EQ
OUT 34.09  ; Z10
LD TR0
CMP(20) DM8 #11  ; 自动车位
AND P_EQ
OUT 34.10  ; Z11
LD TR0
CMP(20) DM8 #12  ; 自动车位
AND P_EQ
OUT 34.12  ; Z12
LD TR0
AND P_GT
OUT 35.15  ; > 12

